TYPE ST_EbaraEVA EXTENDS ST_RoughPump:
STRUCT

(* Output *)
    //q_xRunDO 	:	BOOL; in Rough PUMP


(* Input *)
{attribute 'pytmc' := '
    pv: REMOTE;
    field: ZNAM FALSE;
    field: ONAM TRUE;
    io: io;
    '}
    q_xRemote	:	BOOL;
    {attribute 'pytmc' := '
    pv: ALARM_OK;
    field: ZNAM FALSE;
    field: ONAM TRUE;
    io: i
    '}
    i_xAlarmOK	:	BOOL;

    {attribute 'pytmc' := '
    pv: RUN_DI;
    field: ZNAM FALSE;
    field: ONAM TRUE;
    io: i
    '}
    i_xIsRun		:	BOOL;



END_STRUCT
END_TYPE

(* stored: Version 1.1.0.1, ProductVersion 3.1.4022.18
   DUT ST_EbaraEVA: Id {825d9563-9766-45be-b4c4-16a1335c1e21} *)
